(* IEC 61131-3 sources: tankvalve/src/Valve Class, 3 files *)

(* ---- Valve.st ---- *)
NAMESPACE TankValvelib
    TYPE
        ValveState : (Opened, Closed, Undefined, Error) := Closed;
    END_TYPE
    CLASS PUBLIC Valve IMPLEMENTS IValve
        VAR
         _valveState:BOOL;
        END_VAR

        METHOD PUBLIC Open
            _valveState:=TRUE;
        END_METHOD

        METHOD PUBLIC Close
            _valveState:=FALSE;
            ;
        END_METHOD

        METHOD PUBLIC GetState : ValveState
            IF _valveState THEN
                GetState:=ValveState#Opened;
            ELSE
                GetState:=ValveState#Closed;
            END_IF;
            ;
        END_METHOD

        METHOD PUBLIC WriteCyclic
            VAR_OUTPUT
                valveState:BOOL;
            END_VAR
            valveState:=_valveState;
            ;
        END_METHOD

    END_CLASS

END_NAMESPACE

(* ---- AlwaysOFFValve.st ---- *)
NAMESPACE TankValveLib

    ///常闭阀门类，实现阀门接口
    CLASS PUBLIC AlwaysOFFValve IMPLEMENTS IValve
        ///私有内部变量存储阀门状态
        VAR
        _valveState:BOOL;
        END_VAR

        ///打开，触电断开
        METHOD PUBLIC Open
            _valveState := FALSE;
        END_METHOD

        ///关闭，触电吸合
        METHOD PUBLIC Close
            _valveState:=TRUE;
        END_METHOD

        ///获取阀门状态，返回枚举值
        METHOD PUBLIC GetState:ValveState
            if(_valveState) Then
                GetState:=ValveState#Closed;
            ELSE
                GetState:=ValveState#Opened;
            END_IF;
        END_METHOD

        ///输出Q区
        METHOD PUBLIC WriteCyclic
            VAR_OUTPUT
                outPutSignal:BOOL;
            END_VAR
            outPutSignal:=_valveState;
        END_METHOD
    END_CLASS

END_NAMESPACE

(* ---- ValveWithSensor.st ---- *)
NAMESPACE TankValveLib

    /// 带反馈的阀门类，继承Valve-
    CLASS PUBLIC ValveWithSensor EXTENDS Valve
        VAR PRIVATE
        _closeSensor:BOOL;
        END_VAR
        //扩展方法：读取传感器反馈信号
        METHOD PUBLIC ReadSensor
            VAR_INPUT
                closeSensor : BOOL;
            END_VAR
            _closeSensor := closeSensor;
        END_METHOD

        //重写方法：修改父类Valve的获取状态
        METHOD PUBLIC OVERRIDE GetState : ValveState
            IF (_closeSensor) THEN
                GetState := ValveState#Closed;
            ELSE
                GetState := ValveState#Opened;
            END_IF;
        END_METHOD

    END_CLASS

END_NAMESPACE
